TYPE "MatCountHMI"
VERSION : 0.1
// Block: MatCountHMI
   STRUCT
      PbFAKCalculation : Bool;
      PbFAKDefault : Bool;
      PbFAKPrevious : Bool;
      FAKSetDefaultDone : Bool;
      FAKCalcDone : Bool;
      FAKSetPrevDone : Bool;
      LenghtDesired : LReal;
      LenghtMeasured : LReal;
      FAKPrevious : LReal;
   END_STRUCT;

END_TYPE
